SUBAPPLICATION TOGGLE_RPC_MERGE_QXA_OPC (* 1-Richtungs-Ausgang, klick-toggle statt tastend: ein per OPC-UA-Methodenaufruf (CREATE_METHOD/SERVER_0) empfangener Trigger taktet ein lokales AX_T_FF (Toggle-Flipflop) - dessen Zustand wird per AX_OR_2 mit dem bestehenden IO-Test-Kommando (Remote-Subscribe, gleiches Muster wie MERGE_SWITCH_1_QXA_OPC) zusammengefuehrt. Ausgang treibt den physischen logiBUS-Kanal UND meldet seinen Zustand sowohl an die bestehende IO-Test-Ueberwachung als auch an die echte Funktions-Rueckmeldung (z.B. GreenWhiteBackground am SoftKey, per lokalem Publish + Remote-Subscribe wie bei allen anderen Funktionen dieses Projekts - NICHT per aktivem Client-Write wie im urspruenglichen Uebungs-Vorbild, fuer Konsistenz mit ILOCK_SWITCH_2_QXA_OPC/MERGE_SWITCH_1_QXA_OPC). Fuer echte Klick-Toggle-Funktionen (z.B. Blitzlicht: 1x druecken AN, nochmal druecken AUS) statt tastender Doppelwirkungs-/Einzelausgaenge. *)
  (* Standard: 61499-2; Description: Copyright (c) 2026 Meisterschulen am Ostbahnhof This program and the accompanying materials are made available under the terms of the Eclipse Public License 2.0 which is available at https://www.eclipse.org/legal/epl-2.0/ SPDX-License-Identifier: EPL-2.0 *)
  (* Version 1.1, 2026-09-09, Franz Höpfinger, Meisterschulen am Ostbahnhof, Fix: TRIGGER_SERVER.RSP war nie verdrahtet - blockierte den OPC-UA-Server-Thread bis zu 4s pro Aufruf (haelt open62541s globalen serviceMutex), verzoegerte dadurch JEDE OPC-UA-Statusmeldung projektweit. IND->RSP direkt verdrahtet (argumentloser Trigger, kein CNF noetig). Siehe OPC_UA_VERNETZUNG.md Punkt 12. *)
  (* Version 1.0, 2026-09-07, Franz Höpfinger, Meisterschulen am Ostbahnhof, initial API and implementation and/or initial documentation - Klick-Toggle-Analogon zu MERGE_SWITCH_1_QXA_OPC, RPC-Trigger (SERVER_0/AX_T_FF) statt Pegel-Subscribe als echte Funktionsquelle *)
  PACKAGE MyLib::sys;
  IMPORT logiBUS::io::DQ::logiBUS_DO;
  IMPORT logiBUS::io::DQ::logiBUS_DO_S;
  (* Documentation:
  Klick-Toggle-Ausgang: RPC-Trigger ODER IO-Test
   Fuer Funktionen, die per einmaligem Tastendruck EIN/AUS schalten (Klick-Toggle, z.B. Blitzlicht) statt gehalten zu werden (tastend). Ein SoftKey-Tastendruck (Release-Event) auf dem Bedienmodul loest per CLIENT_0/SERVER_0 einen argumentlosen RPC-Methodenaufruf aus (kein Wertwechsel-Trick, kein Polling noetig - siehe Softkey_Toggle_RPC_TO_Remote_BG_OPC fuer die Bedienmodul-Seite), der hier lokal ein AX_T_FF (Toggle-Flipflop) taktet.
   Der Flipflop-Zustand wird per AX_OR_2 mit dem bestehenden IO-Test-Kommando zusammengefuehrt (IO-Test bleibt nutzbar) und treibt den physischen Ausgang. Wie bei MERGE_SWITCH_1_QXA_OPC/ILOCK_SWITCH_2_QXA_OPC bekommt der resultierende Zustand ZWEI eigene, von den jeweiligen Kommando-Knoten getrennte Rueckmelde-Knoten (ID_TEST_WRITE fuer IO-Diag, ID_STATE_WRITE fuer die echte Funktions-Rueckmeldung) - niemals denselben Knoten wie die zugehoerige Kommando-Adresse, sonst Selbstlatch (siehe OPC_UA_VERNETZUNG.md Punkt 10+11).
   Abweichend vom urspruenglichen Uebungs-Vorbild (Toggle_RPC_FROM_Remote_QXA_OPC, 4diac_training1) wird der Zustand hier NICHT aktiv per CLIENT_1_0 ans Bedienmodul zurueckgeschrieben, sondern lokal publiziert und vom Bedienmodul remote abonniert - konsistent mit allen anderen Funktionen dieses Projekts (Lenkdeichsel, Achslenkung, Hangausgleich).
  *)
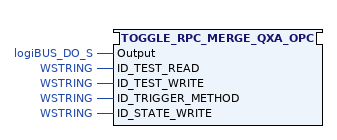
  VAR_INPUT
    Output : logiBUS::io::DQ::logiBUS_DO_S := logiBUS_DO::Invalid; (* Physischer Ausgang *)
    ID_TEST_READ : WSTRING; (* Bestehende IO-Test-Subscribe-Adresse (z.B. STG5_Q0x_READ) *)
    ID_TEST_WRITE : WSTRING; (* Bestehende IO-Test-Publish-Adresse (z.B. STG5_Q0x_WRITE) - EIGENER Knoten, NICHT ID_TEST_READs Knoten (sonst Selbstrueckkopplung/Latch, siehe OPC_UA_VERNETZUNG.md Punkt 10+11) *)
    ID_TRIGGER_METHOD : WSTRING; (* Lokale Methodenadresse (ACTION=CREATE_METHOD) fuer den argumentlosen Toggle-Trigger, wird vom Bedienmodul per CALL_METHOD aufgerufen *)
    ID_STATE_WRITE : WSTRING; (* Lokale Publish-Adresse (ACTION=WRITE) fuer den tatsaechlichen Toggle-Zustand - wird vom Bedienmodul remote abonniert (z.B. fuer GreenWhiteBackground) *)
  END_VAR
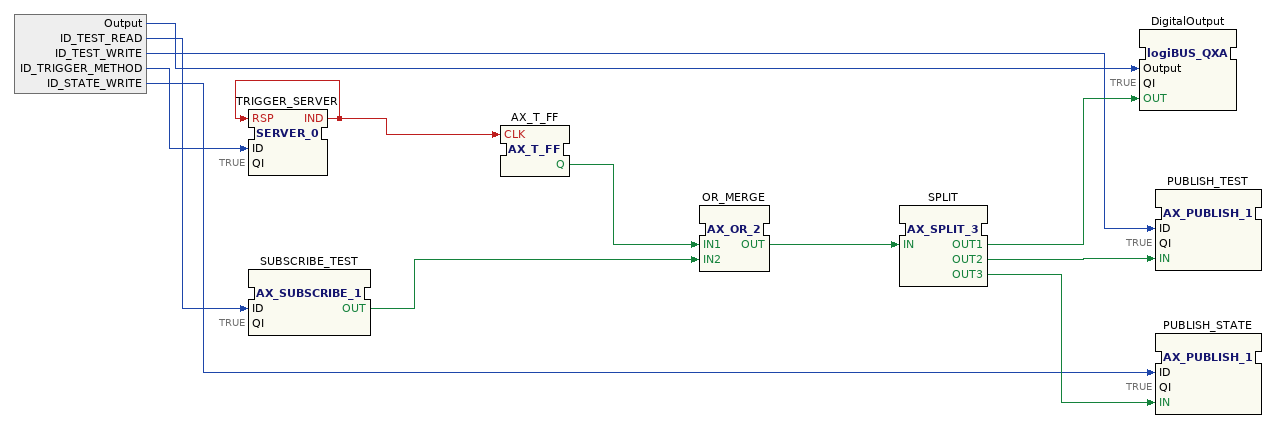
  FBS
    TRIGGER_SERVER : iec61499::net::SERVER_0(QI := TRUE);
    AX_T_FF : adapter::events::unidirectional::AX_T_FF;
    SUBSCRIBE_TEST : adapter::net::AX_SUBSCRIBE_1(QI := TRUE);
    OR_MERGE : adapter::booleanOperators::AX_OR_2;
    DigitalOutput : logiBUS::io::DQ::logiBUS_QXA(QI := TRUE);
    SPLIT : adapter::events::unidirectional::AX_SPLIT_3;
    PUBLISH_TEST : adapter::net::AX_PUBLISH_1(QI := TRUE);
    PUBLISH_STATE : adapter::net::AX_PUBLISH_1(QI := TRUE);
  END_FBS
  EVENT_CONNECTIONS
    TRIGGER_SERVER.IND TO AX_T_FF.CLK;
    TRIGGER_SERVER.IND TO TRIGGER_SERVER.RSP;
  END_CONNECTIONS
  DATA_CONNECTIONS
    Output TO DigitalOutput.Output;
    ID_TEST_READ TO SUBSCRIBE_TEST.ID;
    ID_TEST_WRITE TO PUBLISH_TEST.ID;
    ID_TRIGGER_METHOD TO TRIGGER_SERVER.ID;
    ID_STATE_WRITE TO PUBLISH_STATE.ID;
  END_CONNECTIONS
  ADAPTER_CONNECTIONS
    AX_T_FF.Q TO OR_MERGE.IN1;
    SUBSCRIBE_TEST.OUT TO OR_MERGE.IN2;
    OR_MERGE.OUT TO SPLIT.IN;
    SPLIT.OUT1 TO DigitalOutput.OUT;
    SPLIT.OUT2 TO PUBLISH_TEST.IN;
    SPLIT.OUT3 TO PUBLISH_STATE.IN;
  END_CONNECTIONS
END_SUBAPPLICATION
